# EPICS autosave request: src/iocdoc/testfiles/iocBoot/ioc495idc/auto_positions.req
$(P)m1.DVAL
$(P)m2.DVAL
$(P)m3.DVAL
$(P)m4.DVAL
$(P)m5.DVAL
$(P)m6.DVAL
$(P)m7.DVAL
$(P)m8.DVAL
$(P)m9.DVAL
$(P)m10.DVAL
$(P)m11.DVAL
$(P)m12.DVAL
$(P)m13.DVAL
$(P)m14.DVAL
$(P)m15.DVAL
$(P)m16.DVAL
$(P)m19.DVAL
$(P)m20.DVAL

$(P)sm1.DVAL
$(P)sm2.DVAL
$(P)sm3.DVAL
$(P)sm4.DVAL
$(P)sm5.DVAL
$(P)sm6.DVAL
$(P)sm7.DVAL
$(P)sm8.DVAL
$(P)sm9.DVAL
$(P)sm10.DVAL
$(P)sm11.DVAL
$(P)sm12.DVAL
$(P)sm13.DVAL
$(P)sm14.DVAL
$(P)sm15.DVAL
$(P)sm16.DVAL
$(P)sm17.DVAL
$(P)sm18.DVAL
$(P)sm19.DVAL
$(P)sm20.DVAL
$(P)sm21.DVAL
$(P)sm22.DVAL
$(P)sm23.DVAL
$(P)sm24.DVAL
$(P)sm25.DVAL
$(P)sm26.DVAL
$(P)sm27.DVAL
$(P)sm28.DVAL
$(P)sm29.DVAL
$(P)sm30.DVAL
$(P)sm31.DVAL
$(P)sm32.DVAL
$(P)sm33.DVAL
$(P)sm34.DVAL
$(P)sm35.DVAL
$(P)sm36.DVAL
$(P)sm37.DVAL
$(P)sm38.DVAL
$(P)sm39.DVAL
$(P)sm40.DVAL
$(P)sm40.DVAL
$(P)sm41.DVAL
$(P)sm42.DVAL
$(P)sm43.DVAL
$(P)sm44.DVAL
$(P)sm45.DVAL
$(P)sm46.DVAL
$(P)sm47.DVAL
$(P)sm48.DVAL
$(P)sm49.DVAL
$(P)sm50.DVAL
